// TIA Portal V19 export
DATA_BLOCK "DB_AnalogInput"   // DB11
{ S7_Optimized_Access := 'TRUE'; DB_Accessible_From_OPC_UA := 'FALSE' }
// stored: AutoNumber false, DBAccessibleFromOPCUA false, DBAccessibleFromWebserver false, MemoryReserve 100
   VAR
      ConvertResult { ExternalAccessible := 'False'; ExternalVisible := 'False'; ExternalWritable := 'False'} : "stResult";
   END_VAR
BEGIN
END_DATA_BLOCK
